FUNCTION outputFBD : INT
VAR_INPUT
END_VAR
VAR
	bottomBeltLeft_OB: BOOL;
END_VAR
VAR // added by the converter: edge detectors and wires of the graphical bodies
    _w1 : BOOL;
END_VAR

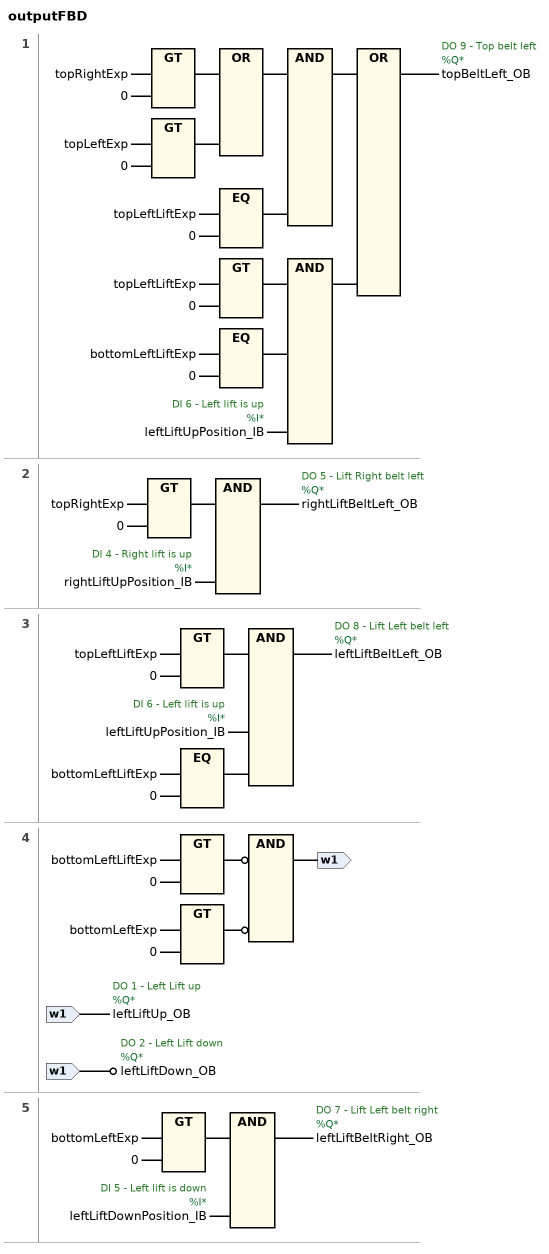
// NETWORK 1
//   leftLiftUpPosition_IB: DI 6 - Left lift is up | AT %I*
//   topBeltLeft_OB: DO 9 - Top belt left | AT %Q*
topBeltLeft_OB := (topRightExp > 0 OR topLeftExp > 0) AND topLeftLiftExp = 0 OR topLeftLiftExp > 0 AND bottomLeftLiftExp = 0 AND leftLiftUpPosition_IB;

// NETWORK 2
//   rightLiftUpPosition_IB: DI 4 - Right lift is up | AT %I*
//   rightLiftBeltLeft_OB: DO 5 - Lift Right belt left | AT %Q*
rightLiftBeltLeft_OB := topRightExp > 0 AND rightLiftUpPosition_IB;

// NETWORK 3
//   leftLiftUpPosition_IB: DI 6 - Left lift is up | AT %I*
//   leftLiftBeltLeft_OB: DO 8 - Lift Left belt left | AT %Q*
leftLiftBeltLeft_OB := topLeftLiftExp > 0 AND leftLiftUpPosition_IB AND bottomLeftLiftExp = 0;

// NETWORK 4
//   leftLiftUp_OB: DO 1 - Left Lift up | AT %Q*
//   leftLiftDown_OB: DO 2 - Left Lift down | AT %Q*
_w1 := NOT (bottomLeftLiftExp > 0) AND NOT (bottomLeftExp > 0);
leftLiftUp_OB := _w1;
leftLiftDown_OB := NOT _w1;

// NETWORK 5
//   leftLiftDownPosition_IB: DI 5 - Left lift is down | AT %I*
//   leftLiftBeltRight_OB: DO 7 - Lift Left belt right | AT %Q*
leftLiftBeltRight_OB := bottomLeftExp > 0 AND leftLiftDownPosition_IB;

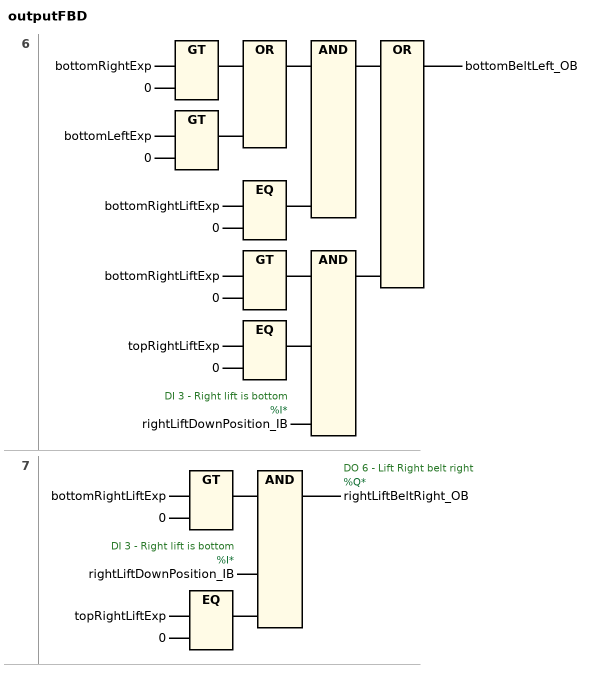
// NETWORK 6
//   rightLiftDownPosition_IB: DI 3 - Right lift is bottom | AT %I*
bottomBeltLeft_OB := (bottomRightExp > 0 OR bottomLeftExp > 0) AND bottomRightLiftExp = 0 OR bottomRightLiftExp > 0 AND topRightLiftExp = 0 AND rightLiftDownPosition_IB;

// NETWORK 7
//   rightLiftDownPosition_IB: DI 3 - Right lift is bottom | AT %I*
//   rightLiftBeltRight_OB: DO 6 - Lift Right belt right | AT %Q*
rightLiftBeltRight_OB := bottomRightLiftExp > 0 AND rightLiftDownPosition_IB AND topRightLiftExp = 0;

END_FUNCTION

(* stored: Version 1.1.0.1, ProductVersion 3.1.4018.5
   POU outputFBD: Id {1331bcc3-23a3-4ead-8e70-3c42710235a2}, SpecialFunc None *)
